Yaskawa INFORM job: R1_BATMAN(-70,-90).JBI

/JOB
//NAME R1_BATMAN(-70,-90)
//POS
///NPOS 78,78,0,2,0,0
///TOOL 0
///POSTYPE PULSE
///PULSE
C00000=29960,139157,41546,-12188,94395,86333
C00001=5087,113588,45388,-11537,82776,83583
C00002=-93778,11955,60659,-8947,36592,72651
C00003=-93780,11950,60654,-8946,36592,72650
C00004=-93781,11948,60652,-8945,36592,72649
C00005=-93780,11939,60644,-8946,36593,72650
C00006=-93781,11938,60643,-8945,36593,72649
C00007=-93780,11939,60644,-8946,36593,72650
C00008=-93781,11948,60652,-8945,36592,72649
C00009=-93785,11949,60653,-8944,36592,72647
C00010=-93785,11947,60651,-8944,36592,72647
C00011=-93785,11949,60653,-8944,36592,72647
C00012=-93781,11948,60652,-8945,36592,72649
C00013=-89364,-8679,43175,-10801,37206,74685
C00014=-88884,-10409,41847,-11019,37191,74917
C00015=-89364,-8679,43175,-10801,37206,74685
C00016=-93780,11939,60644,-8946,36593,72650
C00017=-93779,11942,60646,-8946,36593,72650
C00018=-93776,11947,60651,-8947,36593,72652
C00019=-93769,2183,43640,-18296,65866,26195
C00020=-93777,11958,60661,-19147,60688,27072
C00021=-93780,11952,60656,-19147,60688,27071
C00022=-93780,11950,60653,-19147,60688,27071
C00023=-93432,10219,57502,-18939,61752,27004
C00024=-92881,10084,58322,-18996,61317,27270
C00025=-93783,11955,60658,-19147,60687,27070
C00026=-93782,11957,60660,-19147,60687,27071
C00027=-93780,11963,60666,-19147,60687,27071
C00028=-93777,11953,60656,-8333,71131,73543
C00029=-93779,11947,60651,-8333,71131,73543
C00030=-93780,11945,60649,-8333,71131,73542
C00031=-93411,13542,61674,-8251,71352,73640
C00032=-93498,10227,57484,-8230,72210,73554
C00033=-93781,11950,60654,-12981,71164,71139
C00034=-93788,11963,60666,-12982,71162,71137
C00035=-93787,11966,60668,-12982,71162,71137
C00036=-93785,11972,60674,-12982,71162,71138
C00037=-93790,11982,60683,-12983,71161,71136
C00038=-93792,11976,60678,-12983,71161,71136
C00039=-93793,11973,60675,-12983,71161,71136
C00040=-93287,13524,61710,-12869,71386,71267
C00041=-93445,10242,57524,-12840,72233,71127
C00042=-93800,11989,60690,-12985,71159,71133
C00043=-93799,11991,60692,-12985,71159,71134
C00044=-93798,11997,60698,-12984,71159,71134
C00045=-92523,4991,54420,-21378,64231,23661
C00046=-93035,7669,56779,-21453,64047,23523
C00047=-93234,8762,57755,-21484,63966,23471
C00048=-92881,7098,54706,-21270,64999,23391
C00049=-92314,6971,55534,-21296,64588,23663
C00050=-93800,11991,60692,-21578,63702,23331
C00051=-93799,11994,60694,-21578,63702,23331
C00052=-93797,12000,60700,-21578,63702,23331
C00053=-93779,11959,60662,-15391,75707,-18818
C00054=-93782,11955,60659,-15392,75706,-18819
C00055=-93783,11954,60657,-15392,75706,-18819
C00056=-93511,10386,57641,-15260,76765,-18870
C00057=-94230,9238,56828,-15451,76562,-19066
C00058=-93785,11960,60663,-22039,74213,-17711
C00059=-93788,11966,60669,-22039,74212,-17712
C00060=-93787,11968,60671,-22039,74212,-17711
C00061=-93784,11973,60675,-22038,74213,-17711
C00062=-93787,11968,60670,-16733,84415,-38761
C00063=-93790,11964,60667,-16734,84415,-38762
C00064=-93791,11962,60665,-16734,84414,-38762
C00065=-94303,12956,60893,-16911,84680,-38953
C00066=-93442,10234,57516,-16591,85483,-38802
C00067=-93793,11967,60670,-16735,84414,-38763
C00068=-93792,11969,60671,-16735,84414,-38763
C00069=-93789,11973,60675,-16734,84414,-38762
C00070=-93783,11966,60669,-10361,76115,-17611
C00071=-93786,11962,60665,-10362,76115,-17612
C00072=-93788,11961,60664,-10362,76115,-17612
C00073=-94457,10596,58108,-10503,76898,-17880
C00074=-93439,10231,57514,-10231,77186,-17597
C00075=-93789,11965,60668,-10363,76114,-17612
C00076=-93788,11966,60669,-10363,76114,-17612
C00077=-93785,11970,60672,-10362,76115,-17611
BC00000=68533,13783,1075157
BC00001=67053,15036,1061279
BC00002=199547,17717,1006114
BC00003=197681,18521,980130
BC00004=196934,18842,969737
BC00005=184906,18876,969495
BC00006=184922,19665,961919
BC00007=184906,18876,969495
BC00008=196934,18842,969737
BC00009=203657,27615,944031
BC00010=201268,27622,943983
BC00011=203657,27615,944031
BC00012=196934,18842,969737
BC00013=209489,15,946874
BC00014=209488,15,944109
BC00015=209489,15,946874
BC00016=184906,18876,969495
BC00017=185652,18554,979888
BC00018=187518,17750,1005872
BC00019=202015,16790,1075175
BC00020=202015,16790,1009573
BC00021=198538,19689,987618
BC00022=197148,20849,978836
BC00023=197148,20849,978836
BC00024=197148,20849,978836
BC00025=206805,27229,967131
BC00026=208196,26069,975913
BC00027=211672,23170,997868
BC00028=195363,100167,1007486
BC00029=191913,96802,986312
BC00030=190533,95456,977842
BC00031=190533,95456,977842
BC00032=190533,95456,977842
BC00033=199250,90952,972016
BC00034=223976,67028,942040
BC00035=225644,68183,950262
BC00036=229814,71070,970816
BC00037=248382,93192,948571
BC00038=244212,90305,928017
BC00039=242544,89150,919796
BC00040=242544,89150,919796
BC00041=242544,89150,919796
BC00042=272125,60528,883934
BC00043=273793,61683,892156
BC00044=277963,64570,912710
BC00045=233300,15,972780
BC00046=229823,15,950825
BC00047=228433,15,942043
BC00048=228433,15,942043
BC00049=228433,15,942043
BC00050=275282,27385,885750
BC00051=276672,26225,894532
BC00052=280149,23326,916486
BC00053=205957,59032,1001807
BC00054=205961,58583,974970
BC00055=205963,58403,964235
BC00056=205963,58403,964235
BC00057=205963,58403,964235
BC00058=215521,49805,957546
BC00059=228104,18868,942131
BC00060=228374,18824,952845
BC00061=229049,18715,979629
BC00062=228081,88935,952893
BC00063=227610,85489,928921
BC00064=227422,84110,919332
BC00065=227422,84110,919332
BC00066=227422,84110,919332
BC00067=236678,87321,908192
BC00068=236866,88699,917781
BC00069=237336,92146,941752
BC00070=220067,73521,978437
BC00071=220555,72961,951675
BC00072=220750,72737,940970
BC00073=220750,72737,940970
BC00074=220750,72737,940970
BC00075=228479,91067,931771
BC00076=228284,91290,942476
BC00077=227796,91850,969237
///POSTYPE BASE
///RECTAN
///RCONF 0,0,0,0,1,0,0,0,0,0,0,0,0,0,0,0,0,0,0,0,0,0,0,0
P00006=2.006,1.622,-0.565,0.0000,0.0000,0.0000
P00021=0.073,2.058,-0.109,0.0000,0.0000,0.0000
//INST
///DATE 2023/11/17 10:25
///ATTR SC,RW
///GROUP1 RB1,BS1
NOP
'R1_BATMAN(-70,-90)
'Path S1475
SFTOF
MOVJ C00000 BC00000 VJ=40.00
CALL JOB:CLEAN-R1_LONG
MOVJ C00001 BC00001 VJ=40.00
MOVJ C00002 BC00002 VJ=15.00
MOVJ C00003 BC00003 VJ=15.00
MOVL C00004 BC00004 V=100.0
MOVL C00005 BC00005 V=60.0
REFP 3 C00006 BC00006
CALL JOB:SEARCH-R1
SET P021 P006
SFTON P021
MOVL C00007 BC00007 V=60.0
MOVL C00008 BC00008 V=100.0
MOVL C00009 BC00009 V=60.0
REFP 3 C00010 BC00010
CALL JOB:SEARCH-R1
SET P021 P006
SFTON P021
MOVL C00011 BC00011 V=60.0
MOVL C00012 BC00012 V=100.0
MOVL C00013 BC00013 V=60.0
REFP 3 C00014 BC00014
CALL JOB:SEARCH-R1
SET P021 P006
SFTON P021
MOVL C00015 BC00015 V=60.0
MOVL C00016 BC00016 V=100.0
MOVL C00017 BC00017 V=100.0
MOVL C00018 BC00018 V=166.7
'Path W1468
SFTOF
SFTON P021
MOVJ C00019 BC00019 VJ=15.00
MOVJ C00020 BC00020 VJ=15.00
MOVJ C00021 BC00021 VJ=15.00
MOVL C00022 BC00022 V=100.0 PL=0
REFP 1 C00023 BC00023
REFP 2 C00024 BC00024
MACRO1 MJ#(0) ARGF0
ARCON
MOVL C00025 BC00025 V=10.0
ARCOF
MOVL C00026 BC00026 V=100.0
MOVL C00027 BC00027 V=166.7
SFTOF
'Path W1469
SFTOF
SFTON P021
MOVJ C00028 BC00028 VJ=15.00
MOVJ C00029 BC00029 VJ=15.00
MOVL C00030 BC00030 V=100.0 PL=0
REFP 1 C00031 BC00031
REFP 2 C00032 BC00032
MACRO1 MJ#(0) ARGF0
ARCON
MOVL C00033 BC00033 V=10.0
MOVL C00034 BC00034 V=10.0
ARCOF
MOVL C00035 BC00035 V=100.0
MOVL C00036 BC00036 V=166.7
SFTOF
'Path W1470
SFTOF
SFTON P021
MOVJ C00037 BC00037 VJ=15.00
MOVJ C00038 BC00038 VJ=15.00
MOVL C00039 BC00039 V=100.0 PL=0
REFP 1 C00040 BC00040
REFP 2 C00041 BC00041
MACRO1 MJ#(0) ARGF0
ARCON
MOVL C00042 BC00042 V=10.0
ARCOF
MOVL C00043 BC00043 V=100.0
MOVL C00044 BC00044 V=166.7
SFTOF
'Path W1471
SFTOF
SFTON P021
MOVJ C00045 BC00045 VJ=15.00
MOVJ C00046 BC00046 VJ=15.00
MOVL C00047 BC00047 V=100.0 PL=0
REFP 1 C00048 BC00048
REFP 2 C00049 BC00049
MACRO1 MJ#(0) ARGF0
ARCON
MOVL C00050 BC00050 V=10.0
ARCOF
MOVL C00051 BC00051 V=100.0
MOVL C00052 BC00052 V=166.7
SFTOF
'Path W1472
SFTOF
SFTON P021
MOVJ C00053 BC00053 VJ=15.00
MOVJ C00054 BC00054 VJ=15.00
MOVL C00055 BC00055 V=100.0 PL=0
REFP 1 C00056 BC00056
REFP 2 C00057 BC00057
MACRO1 MJ#(0) ARGF0
ARCON
MOVL C00058 BC00058 V=10.0
MOVL C00059 BC00059 V=10.0
ARCOF
MOVL C00060 BC00060 V=100.0
MOVL C00061 BC00061 V=166.7
SFTOF
'Path W1473
SFTOF
SFTON P021
MOVJ C00062 BC00062 VJ=15.00
MOVJ C00063 BC00063 VJ=15.00
MOVL C00064 BC00064 V=100.0 PL=0
REFP 1 C00065 BC00065
REFP 2 C00066 BC00066
MACRO1 MJ#(0) ARGF0
ARCON
MOVL C00067 BC00067 V=10.0
ARCOF
MOVL C00068 BC00068 V=100.0
MOVL C00069 BC00069 V=166.7
SFTOF
'Path W1474
SFTOF
SFTON P021
MOVJ C00070 BC00070 VJ=15.00
MOVJ C00071 BC00071 VJ=15.00
MOVL C00072 BC00072 V=100.0 PL=0
REFP 1 C00073 BC00073
REFP 2 C00074 BC00074
MACRO1 MJ#(0) ARGF0
ARCON
MOVL C00075 BC00075 V=10.0
ARCOF
MOVL C00076 BC00076 V=100.0
MOVL C00077 BC00077 V=166.7
SFTOF
END
